FUNCTION_BLOCK TClock IMPLEMENTS IClock
VAR
    _DateTimeInitialised : BOOL; // to detect startup
	_NowAsTimeStruct: TIMESTRUCT;
    
	NT_GetTime1: NT_GetTime;
	TON1: TON;
    GetWindowsTimeRequest : BOOL;
	SyncRequest: BOOL;
    F_TRIG1 : F_TRIG;
	RTC_EX2: RTC_EX2;
	PresetTime: TIMESTRUCT;
    
END_VAR

// Request a sync every 10s
TON1(IN := NOT GetWindowsTimeRequest, PT := T#10S, Q=> GetWindowsTimeRequest);

// Get time from Windows clock
NT_GetTime1(
	NetId := '',
	Start := GetWindowsTimeRequest OR NOT _DateTimeInitialised, // request on first scan also
	TmOut := T#2S,
    Busy => ,
    Err => ,
    ErrId => ,
	TimeStr => PresetTime);

// Request sync to Windows time when time received
F_TRIG1(CLK :=  NT_GetTime1.Busy, Q=> SyncRequest);   
    
// Sync RTC to Windows time
RTC_EX2(
	EN:= SyncRequest, // re-initialise to Windows clock following sync request
	PDT:= PresetTime, // time to sync to
	PMICRO:= PresetTime.wMilliseconds, 
	Q=> , 
	CDT=> _NowAsTimeStruct, // time updated on every call
	CMICRO=> );
    
IF SyncRequest THEN    
    _DateTimeInitialised := TRUE;
END_IF

PROPERTY DateTimeInitialised : BOOL
GET
DateTimeInitialised := _DateTimeInitialised;
END_GET
END_PROPERTY

PROPERTY NowAsDateTime : DT
GET
NowAsDateTime := SYSTEMTIME_TO_DT(TIMESTR:= _NowAsTimeStruct);
END_GET
END_PROPERTY

PROPERTY NowAsTimeStruct : REFERENCE TO TIMESTRUCT
GET
NowAsTimeStruct REF= _NowAsTimeStruct;
END_GET
END_PROPERTY

END_FUNCTION_BLOCK

(* stored: Version 1.1.0.1, ProductVersion 3.1.4024.3
   POU TClock: Id {60fbc1e8-84a6-0a94-1867-c658ee7c5917}, SpecialFunc None
   Property DateTimeInitialised: Id {e8f6a0ac-8cab-0576-20d1-a9d1105d53b1}
   Get Get: Id {42cab26b-3b1d-0bb4-1474-ed41ca44b6a2}
   Property NowAsDateTime: Id {0ac35ca2-8b7a-0a8f-0365-48a1329f4316}
   Get Get: Id {9d4c4446-62c2-0032-2ced-58ccd05c32d6}
   Property NowAsTimeStruct: Id {3bfe5d05-6073-0f86-297a-ba3520cf1017}
   Get Get: Id {381ca9bf-dda6-0e58-115d-884e42c4e40d} *)
